// TIA Portal project "FuncionFC" (V16)

(* hardware
DEVICE "S7-1200 station_1"  S7-1200 Station
   slot 0: "Rack_0"  S7-1200 Rack  Rack  V1.0
   slot 1: "PLC_1"  CPU 1214C AC/DC/Rly  6ES7 214-1BG40-0XB0  V4.4
*)

// ===== PLC "PLC_1"  CPU 1214C AC/DC/Rly =====

VAR_GLOBAL   // PLC tag table "Tabla de variables estándar"
   "START" AT %I0.0 : Bool;
   "S A" AT %I0.1 : Bool;
   "S B" AT %I0.2 : Bool;
   "S C" AT %I0.3 : Bool;
   "S D" AT %I0.4 : Bool;
   "S AB" AT %I0.5 : Bool;
   "S CD" AT %I0.6 : Bool;
   "S ABCD" AT %I0.7 : Bool;
   "EV A" AT %Q1.0 : Bool;
   "EV B" AT %Q1.1 : Bool;
   "EV C" AT %Q1.2 : Bool;
   "EV D" AT %Q1.3 : Bool;
   "EV AB" AT %Q1.4 : Bool;
   "EV DC" AT %Q1.5 : Bool;
   "EV ABCD" AT %Q1.6 : Bool;
END_VAR

// folder: System blocks/Program resources

DATA_BLOCK "IEC_Timer_0_DB"   // DB1
{ S7_Optimized_Access := 'TRUE' }
AUTHOR : Simatic
FAMILY : IEC
NAME : IEC_TMR
VERSION : 1.0
// stored: InstanceOfName IEC_TIMER
"IEC_TIMER"
BEGIN
END_DATA_BLOCK

// folder: (top level)

FUNCTION "1 Producto A" : Void   // FC1, LAD
{ S7_Optimized_Access := 'TRUE' }
VERSION : 0.1
   VAR_INPUT
      START : Bool;
      APAGAR : Bool;
   END_VAR
   VAR_IN_OUT
      ElectroValvula : Bool;
   END_VAR
BEGIN

REGION Network 1: Se agrega acá y no en Output porque necesito feedback
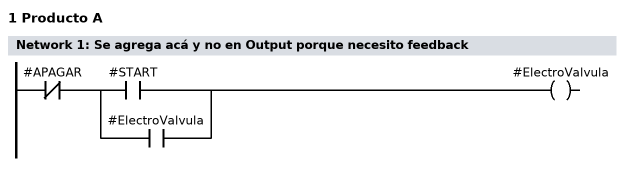
   RUNG wire#powerrail
      I_Contact( #APAGAR )
      wire#w1
      Contact( #START )
      wire#w2
      Coil( #ElectroValvula )
   END_RUNG
   RUNG wire#w1
      Contact( #ElectroValvula )
   END_RUNG wire#w2
   // the same network as SCL:
   #ElectroValvula := NOT #APAGAR AND (#START OR #ElectroValvula);
END_REGION
END_FUNCTION

FUNCTION "2 Producto B" : Void   // FC2, LAD
{ S7_Optimized_Access := 'TRUE' }
VERSION : 0.1
   VAR_INPUT
      ENCENDER : Bool;
      APAGAR : Bool;
   END_VAR
   VAR_IN_OUT
      ElectroValvula : Bool;   // Se agrega acá y no en Output porque necesito feedback
   END_VAR
BEGIN

REGION Network 1: Se agrega acá y no en Output porque necesito feedback
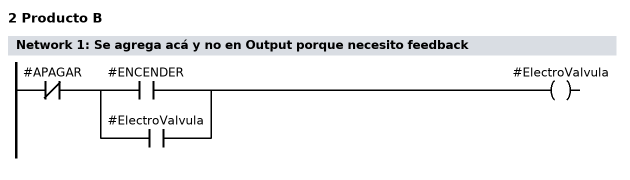
   RUNG wire#powerrail
      I_Contact( #APAGAR )
      wire#w1
      Contact( #ENCENDER )
      wire#w2
      Coil( #ElectroValvula )
   END_RUNG
   RUNG wire#w1
      Contact( #ElectroValvula )
   END_RUNG wire#w2
   // the same network as SCL:
   #ElectroValvula := NOT #APAGAR AND (#ENCENDER OR #ElectroValvula);
END_REGION
END_FUNCTION

FUNCTION "3 Producto C" : Void   // FC3, LAD
{ S7_Optimized_Access := 'TRUE' }
VERSION : 0.1
   VAR_INPUT
      ENCENDER : Bool;
      APAGAR : Bool;
   END_VAR
   VAR_IN_OUT
      ElectroValvula : Bool;   // Se agrega acá y no en Output porque necesito feedback
   END_VAR
BEGIN

REGION Network 1: Se agrega acá y no en Output porque necesito feedback
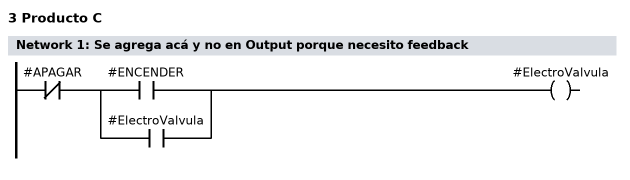
   RUNG wire#powerrail
      I_Contact( #APAGAR )
      wire#w1
      Contact( #ENCENDER )
      wire#w2
      Coil( #ElectroValvula )
   END_RUNG
   RUNG wire#w1
      Contact( #ElectroValvula )
   END_RUNG wire#w2
   // the same network as SCL:
   #ElectroValvula := NOT #APAGAR AND (#ENCENDER OR #ElectroValvula);
END_REGION
END_FUNCTION

FUNCTION "7 Producto ABCD" : Void   // FC4, LAD
{ S7_Optimized_Access := 'TRUE' }
VERSION : 0.1
   VAR_INPUT
      ENCENDER : Bool;
      TIEMPO : Time;
   END_VAR
   VAR_IN_OUT
      ElectroValvula : Bool;   // Se agrega acá y no en Output porque necesito feedback
   END_VAR
BEGIN

REGION Network 1: Se agrega acá y no en Output porque necesito feedback
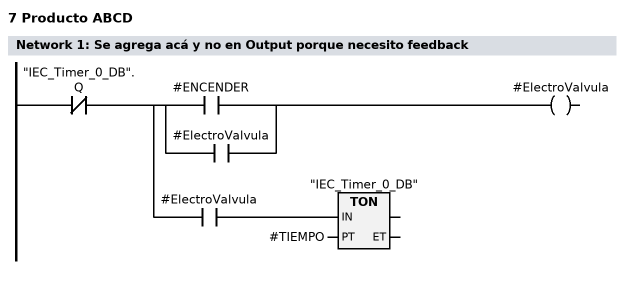
   #ElectroValvula := NOT "IEC_Timer_0_DB".Q AND (#ENCENDER OR #ElectroValvula);
   "IEC_Timer_0_DB".TON(IN := NOT "IEC_Timer_0_DB".Q AND #ElectroValvula, PT := #TIEMPO);
END_REGION
END_FUNCTION

FUNCTION "5 Producto AB" : Void   // FC5, LAD
{ S7_Optimized_Access := 'TRUE' }
VERSION : 0.1
   VAR_INPUT
      ENCENDER : Bool;
      APAGAR : Bool;
   END_VAR
   VAR_IN_OUT
      ElectroValvula : Bool;   // Se agrega acá y no en Output porque necesito feedback
   END_VAR
BEGIN

REGION Network 1: Se agrega acá y no en Output porque necesito feedback
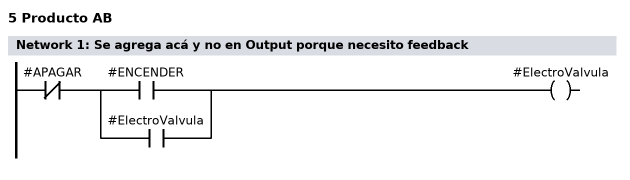
   RUNG wire#powerrail
      I_Contact( #APAGAR )
      wire#w1
      Contact( #ENCENDER )
      wire#w2
      Coil( #ElectroValvula )
   END_RUNG
   RUNG wire#w1
      Contact( #ElectroValvula )
   END_RUNG wire#w2
   // the same network as SCL:
   #ElectroValvula := NOT #APAGAR AND (#ENCENDER OR #ElectroValvula);
END_REGION
END_FUNCTION

FUNCTION "6 Producto CD" : Void   // FC6, LAD
{ S7_Optimized_Access := 'TRUE' }
VERSION : 0.1
   VAR_INPUT
      ENCENDER : Bool;
      APAGAR : Bool;
   END_VAR
   VAR_IN_OUT
      ElectroValvula : Bool;   // Se agrega acá y no en Output porque necesito feedback
   END_VAR
BEGIN

REGION Network 1: Se agrega acá y no en Output porque necesito feedback
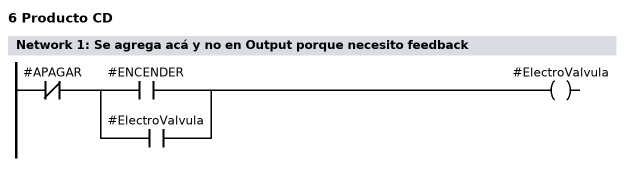
   RUNG wire#powerrail
      I_Contact( #APAGAR )
      wire#w1
      Contact( #ENCENDER )
      wire#w2
      Coil( #ElectroValvula )
   END_RUNG
   RUNG wire#w1
      Contact( #ElectroValvula )
   END_RUNG wire#w2
   // the same network as SCL:
   #ElectroValvula := NOT #APAGAR AND (#ENCENDER OR #ElectroValvula);
END_REGION
END_FUNCTION

FUNCTION "4 Producto D" : Void   // FC7, LAD
{ S7_Optimized_Access := 'TRUE' }
VERSION : 0.1
   VAR_INPUT
      ENCENDER : Bool;
      APAGAR : Bool;
   END_VAR
   VAR_IN_OUT
      ElectroValvula : Bool;   // Se agrega acá y no en Output porque necesito feedback
   END_VAR
BEGIN

REGION Network 1: Se agrega acá y no en Output porque necesito feedback
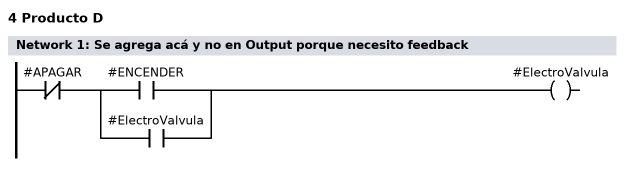
   RUNG wire#powerrail
      I_Contact( #APAGAR )
      wire#w1
      Contact( #ENCENDER )
      wire#w2
      Coil( #ElectroValvula )
   END_RUNG
   RUNG wire#w1
      Contact( #ElectroValvula )
   END_RUNG wire#w2
   // the same network as SCL:
   #ElectroValvula := NOT #APAGAR AND (#ENCENDER OR #ElectroValvula);
END_REGION
END_FUNCTION

ORGANIZATION_BLOCK "Main"   // OB1, LAD, ProgramCycle
TITLE = "Main Program Sweep (Cycle)"
{ S7_Optimized_Access := 'TRUE' }
VERSION : 0.1
   VAR_INPUT
      Initial_Call : Bool;   // Initial call of this OB
      Remanence : Bool;   // =True, if remanent data are available
   END_VAR
BEGIN

REGION Network 1
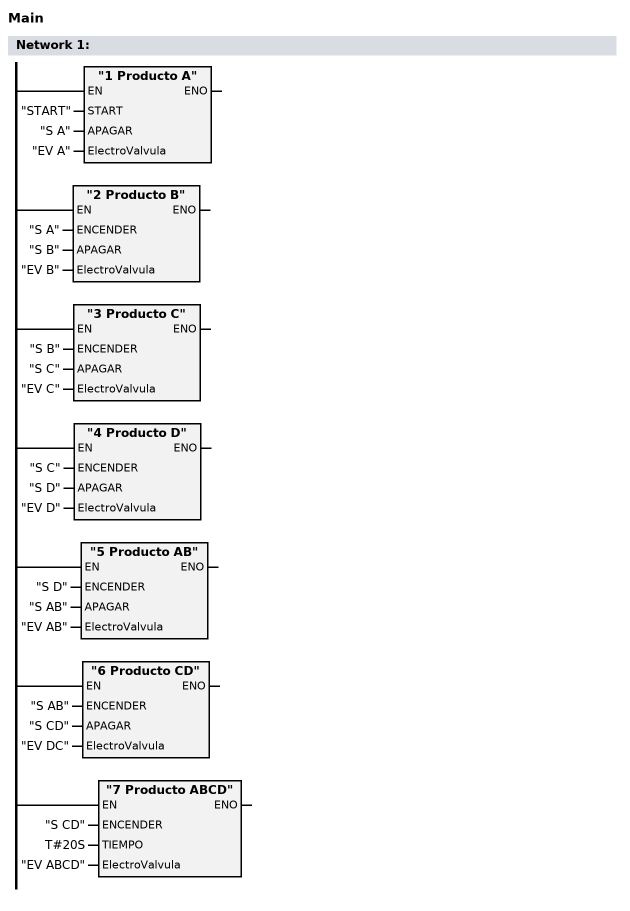
   RUNG wire#powerrail
      "1 Producto A"(START := "START", APAGAR := "S A", ElectroValvula := "EV A")
   END_RUNG
   RUNG wire#powerrail
      "2 Producto B"(ENCENDER := "S A", APAGAR := "S B", ElectroValvula := "EV B")
   END_RUNG
   RUNG wire#powerrail
      "3 Producto C"(ENCENDER := "S B", APAGAR := "S C", ElectroValvula := "EV C")
   END_RUNG
   RUNG wire#powerrail
      "4 Producto D"(ENCENDER := "S C", APAGAR := "S D", ElectroValvula := "EV D")
   END_RUNG
   RUNG wire#powerrail
      "5 Producto AB"(ENCENDER := "S D", APAGAR := "S AB", ElectroValvula := "EV AB")
   END_RUNG
   RUNG wire#powerrail
      "6 Producto CD"(ENCENDER := "S AB", APAGAR := "S CD", ElectroValvula := "EV DC")
   END_RUNG
   RUNG wire#powerrail
      "7 Producto ABCD"(ENCENDER := "S CD", TIEMPO := T#20S, ElectroValvula := "EV ABCD")
   END_RUNG
   // the same network as SCL:
   "1 Producto A"(START := "START", APAGAR := "S A", ElectroValvula := "EV A");
   "2 Producto B"(ENCENDER := "S A", APAGAR := "S B", ElectroValvula := "EV B");
   "3 Producto C"(ENCENDER := "S B", APAGAR := "S C", ElectroValvula := "EV C");
   "4 Producto D"(ENCENDER := "S C", APAGAR := "S D", ElectroValvula := "EV D");
   "5 Producto AB"(ENCENDER := "S D", APAGAR := "S AB", ElectroValvula := "EV AB");
   "6 Producto CD"(ENCENDER := "S AB", APAGAR := "S CD", ElectroValvula := "EV DC");
   "7 Producto ABCD"(ENCENDER := "S CD", TIEMPO := T#20S, ElectroValvula := "EV ABCD");
END_REGION
END_ORGANIZATION_BLOCK